{attribute 'GeneratedUsingTerminal: AT2050-5500-0018'}
{attribute addProperty BoxType "AT2050-5500-0018"}
{attribute addProperty Id "StatusAT %I*UINT2Value_ChannelAT %I*ARRAY[0..31] OF INT64"}
{attribute addProperty CRC "3217050683"}
{attribute addProperty Size "66"}
TYPE FB_Inputs_4BC4AA01 EXTENDS InputBase_8311D824 :
STRUCT
	{attribute addProperty Name "Status"}
	Status AT %I* : UINT;
	{attribute addProperty Name "Value_Channel"}
	Value_Channel AT %I* : ARRAY[0..31] OF INT;
END_STRUCT
END_TYPE

(* stored: Version 1.2.0.0, ProductVersion 3.1.4024.9
   DUT FB_Inputs_4BC4AA01: Id {83830208-0157-4df1-8342-092b4b367be7} *)
